// TIA Portal V20 export
DATA_BLOCK "QDAS_SendBuffer"   // DB302
{ S7_Optimized_Access := 'TRUE' }
// stored: InstanceOfName typeReadVGageProData, InstanceOfType UDT
"typeReadVGageProData"
   // VAR
   //    heartbeatActive : Bool;
   //    dataCollected : Bool;
   //    plcOK : Bool;
   //    spareIn_1 : Bool;
   //    spareIn_2 : Bool;
   //    spareIn_3 : Bool;
   //    spareIn_4 : Bool;
   //    spareIn_5 : Bool;
   // END_VAR
BEGIN
END_DATA_BLOCK
